# B&R Automation Studio project Get_Weather
Automation Studio 4.2.1.211

## Logical view

### WeaTypes.typ
```iecst
TYPE
	weather_typ : 	STRUCT
		temp : REAL;
		humidity : REAL;
		wind_speed : REAL;
		wind_dir : REAL;
		clouds : REAL;
		isValid : BOOL;
	END_STRUCT;
END_TYPE
```

### WeaVariables.var
```iecst
VAR
	weather : weather_typ;
	response_JSON_valid : BOOL;
	response_JSON : STRING[1000];
END_VAR
```

### Program Logical/GetWeather/doHTTP (IEC)

#### Cyclic.fbd - Cyclic code
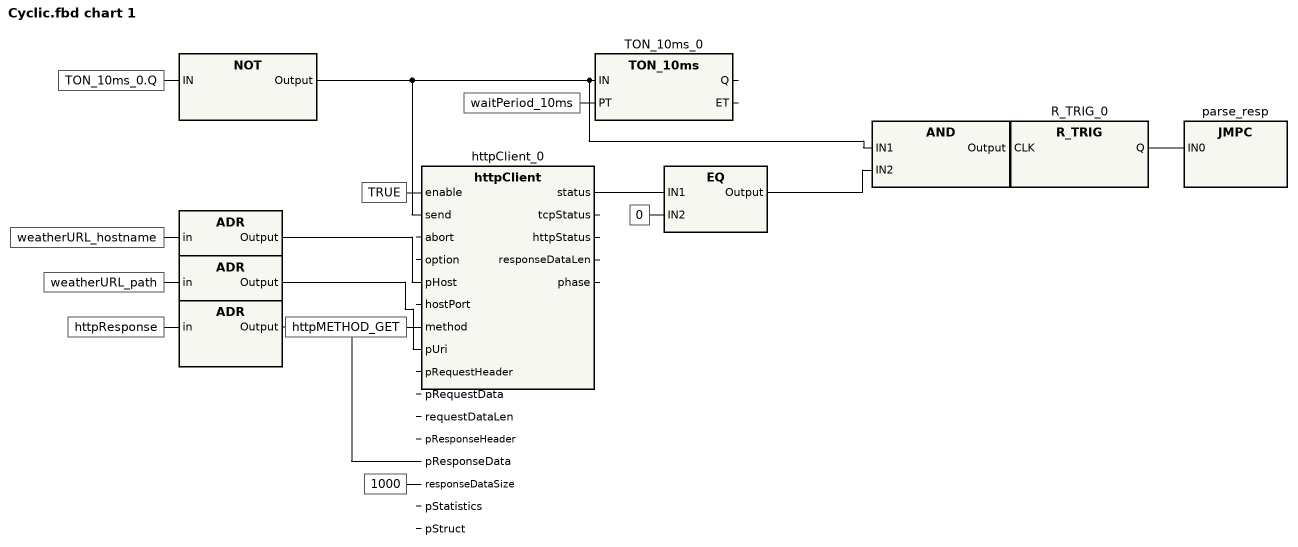
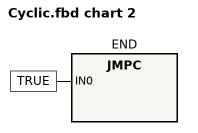
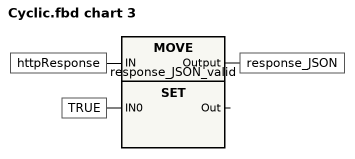
Diagram, in the editor's own instruction-list form stored in the file:
```il
PROGRAM _CYCLIC
VAR
	zz0000FCT_1_1_NOT_Output : ANY;
	zz0000FCT_1_1_ADR_Output : UDINT;
	zz0000FCT_1_2_ADR_Output : UDINT;
	zz0000FCT_1_3_ADR_Output : UDINT;
	zz0000FCT_1_1_EQ_Output : BOOL;
	zz0000FCT_1_1_AND_Output : BOOL;
	zz0000OP_3_1_SET_Out : BOOL;
END_VAR

{NetworkNumber := 1}
LD TON_10ms_0.Q
NOT
ST zz0000FCT_1_1_NOT_Output
LD zz0000FCT_1_1_NOT_Output
ST TON_10ms_0.IN
LD waitPeriod_10ms
ST TON_10ms_0.PT
CAL TON_10ms_0
LD weatherURL_hostname
ADR
ST zz0000FCT_1_1_ADR_Output
LD weatherURL_path
ADR
ST zz0000FCT_1_2_ADR_Output
LD httpResponse
ADR
ST zz0000FCT_1_3_ADR_Output
LD TRUE
ST httpClient_0.enable
LD zz0000FCT_1_1_NOT_Output
ST httpClient_0.send
LD zz0000FCT_1_1_ADR_Output
ST httpClient_0.pHost
LD httpMETHOD_GET
ST httpClient_0.method
LD zz0000FCT_1_2_ADR_Output
ST httpClient_0.pUri
LD zz0000FCT_1_3_ADR_Output
ST httpClient_0.pResponseData
LD 1000
ST httpClient_0.responseDataSize
CAL httpClient_0
LD httpClient_0.status
EQ 0
ST zz0000FCT_1_1_EQ_Output
LD zz0000FCT_1_1_NOT_Output
AND zz0000FCT_1_1_EQ_Output
ST zz0000FCT_1_1_AND_Output
LD zz0000FCT_1_1_AND_Output
ST R_TRIG_0.CLK
CAL R_TRIG_0
LD R_TRIG_0.Q
JMPC parse_resp

{NetworkNumber := 2}
LD TRUE
JMPC END

parse_resp:
{NetworkNumber := 3}
LD httpResponse
MOVE
ST response_JSON
LD TRUE
S response_JSON_valid
LD  response_JSON_valid
ST zz0000OP_3_1_SET_Out

END:
{NetworkNumber := 4}

END_PROGRAM
```

#### Init.fbd - Initialization code
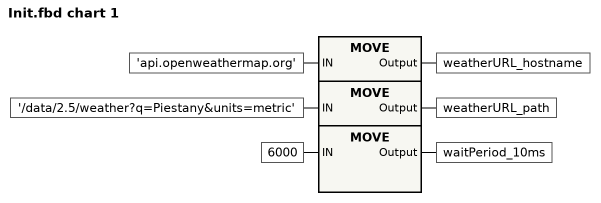
Diagram, in the editor's own instruction-list form stored in the file:
```il
PROGRAM _INIT

{NetworkNumber := 1}
LD 'api.openweathermap.org'
MOVE
ST weatherURL_hostname
LD '/data/2.5/weather?q=Piestany&units=metric'
MOVE
ST weatherURL_path
LD 6000
MOVE
ST waitPeriod_10ms

END_PROGRAM
```

#### Exit.fbd - Exit code
```iecst
PROGRAM _EXIT

(* TODO : Add your code here *)

END_PROGRAM
```

#### GetWheater.var - Local variables
```iecst
VAR
	httpResponse : STRING[1000];
	httpClient_0 : httpClient;
	weatherURL_hostname : STRING[100];
	weatherURL_path : STRING[200];
	TOFF_10ms_0 : TOF_10ms;
	waitPeriod_10ms : UINT;
	R_TRIG_0 : R_TRIG;
	TOF_10ms_0 : TOF_10ms;
	TON_10ms_0 : TON_10ms;
END_VAR
```

### Program Logical/GetWeather/WParser (ANSIC)

#### Cyclic.cpp - Cyclic code
```cpp
#include <bur/plctypes.h>

#ifdef _DEFAULT_INCLUDES
	#include <AsDefault.h>
#endif

#include "jansson.h"

void _CYCLIC ProgramCyclic(void)
{

	if( response_JSON_valid) {
		response_JSON_valid = 0;

		//init structure
		json_t *root;
		json_error_t error;
		root = json_loads(response_JSON, 0, &error);

		if( root) {
			//parse
			/*
			{
			"coord":{"lon":17.75,"lat":48.61},
			"sys":{"message":1.7319,"country":"Slovakia","sunrise":1430623518,"sunset":1430676384},
			"weather":[{"id":500,"main":"Rain","description":"light rain","icon":"10d"}],
			"base":"stations",
			"main":{
			."temp":284.817,
			."temp_min":284.817,
			."temp_max":284.817,
			."pressure":994.66,
			."sea_level":1028.88,
			."grnd_level":994.66,
			."humidity":75},
			"wind":{"speed":3.27,"deg":160.002},
			"clouds":{"all":92},
			"rain":{"3h":0.185},
			"dt":1430646855,
			"id":3056697,
			"name":"Krakovany",
			"cod":200
			}
			*/

			json_t *jmain=json_object_get( root,"main");
			r1=json_unpack(jmain,"{s:F}","temp",&p_temp);
			r2=json_unpack(jmain,"{s:F}","humidity",&p_humidity);

			json_t *jwind=json_object_get( root,"wind");
			r3=json_unpack(jwind,"{s:F}","speed",&p_wind_speed);
			r4=json_unpack(jwind,"{s:F}","deg",&p_wind_deg);

			json_t *jclouds = json_object_get( root,"clouds");
			r5=json_unpack(jclouds,"{s:F}","all",&p_clouds);

			//free
			json_decref(root);

			if( r1+r2+r3+r4+r5 == 0) {
				weather.temp = p_temp;
				weather.clouds = p_clouds;
				weather.wind_dir = p_wind_deg;
				weather.wind_speed = p_wind_speed;
				weather.humidity = p_humidity;
				weather.isValid = 1;
			} else {
				weather.isValid = 0;
			}
		} else { //root not found
			weather.isValid = 0;
		}
	}
}
```

#### Init.cpp - Initialization code
```cpp
#include <bur/plctypes.h>

#ifdef _DEFAULT_INCLUDES
	#include <AsDefault.h>
#endif

void _INIT ProgramInit(void)
{

}
```

#### Exit.cpp - Exit code
```cpp
#include <bur/plctypes.h>

#ifdef _DEFAULT_INCLUDES
	#include <AsDefault.h>
#endif

void _EXIT ProgramExit(void)
{

}
```

#### WParserVar.var - Local variables
```iecst
VAR
	p_humidity : LREAL;
	p_wind_deg : LREAL;
	p_wind_speed : LREAL;
	p_clouds : LREAL;
	r1 : INT;
	r2 : INT;
	r3 : INT;
	r4 : INT;
	r5 : INT;
	p_temp : LREAL;
END_VAR
```

#### hashtable_seed.c
```c
/* Generate sizeof(uint32_t) bytes of as random data as possible to seed
   the hash function.
*/

#ifdef HAVE_CONFIG_H
#include <jansson_private_config.h>
#endif

#include <stdio.h>
#include <time.h>

#ifdef HAVE_STDINT_H
#include <stdint.h>
#endif

#ifdef HAVE_FCNTL_H
#include <fcntl.h>
#endif

#ifdef HAVE_SCHED_H
#include <sched.h>
#endif

#ifdef HAVE_UNISTD_H
#include <unistd.h>
#endif

#ifdef HAVE_SYS_STAT_H
#include <sys/stat.h>
#endif

#ifdef HAVE_SYS_TIME_H
#include <sys/time.h>
#endif

#ifdef HAVE_SYS_TYPES_H
#include <sys/types.h>
#endif

#if defined(_WIN32)
/* For GetModuleHandle(), GetProcAddress() and GetCurrentProcessId() */
#include <windows.h>
#endif

#include "jansson.h"

static uint32_t buf_to_uint32(char *data) {
    size_t i;
    uint32_t result = 0;

    for (i = 0; i < sizeof(uint32_t); i++)
        result = (result << 8) | (unsigned char)data[i];

    return result;
}

/* /dev/urandom */
#if !defined(_WIN32) && defined(USE_URANDOM)
static int seed_from_urandom(uint32_t *seed) {
    /* Use unbuffered I/O if we have open(), close() and read(). Otherwise
       fall back to fopen() */

    char data[sizeof(uint32_t)];
    int ok;

#if defined(HAVE_OPEN) && defined(HAVE_CLOSE) && defined(HAVE_READ)
    int urandom;
    urandom = open("/dev/urandom", O_RDONLY);
    if (urandom == -1)
        return 1;

    ok = read(urandom, data, sizeof(uint32_t)) == sizeof(uint32_t);
    close(urandom);
#else
    FILE *urandom;

    urandom = fopen("/dev/urandom", "rb");
    if (!urandom)
        return 1;

    ok = fread(data, 1, sizeof(uint32_t), urandom) == sizeof(uint32_t);
    fclose(urandom);
#endif

    if (!ok)
        return 1;

    *seed = buf_to_uint32(data);
    return 0;
}
#endif

/* Windows Crypto API */
#if defined(_WIN32) && defined(USE_WINDOWS_CRYPTOAPI)
#include <wincrypt.h>

typedef BOOL (WINAPI *CRYPTACQUIRECONTEXTA)(HCRYPTPROV *phProv, LPCSTR pszContainer, LPCSTR pszProvider, DWORD dwProvType, DWORD dwFlags);
typedef BOOL (WINAPI *CRYPTGENRANDOM)(HCRYPTPROV hProv, DWORD dwLen, BYTE *pbBuffer);
typedef BOOL (WINAPI *CRYPTRELEASECONTEXT)(HCRYPTPROV hProv, DWORD dwFlags);

static int seed_from_windows_cryptoapi(uint32_t *seed)
{
    HINSTANCE hAdvAPI32 = NULL;
    CRYPTACQUIRECONTEXTA pCryptAcquireContext = NULL;
    CRYPTGENRANDOM pCryptGenRandom = NULL;
    CRYPTRELEASECONTEXT pCryptReleaseContext = NULL;
    HCRYPTPROV hCryptProv = 0;
    BYTE data[sizeof(uint32_t)];
    int ok;

    hAdvAPI32 = GetModuleHandle(TEXT("advapi32.dll"));
    if(hAdvAPI32 == NULL)
        return 1;

    pCryptAcquireContext = (CRYPTACQUIRECONTEXTA)GetProcAddress(hAdvAPI32, "CryptAcquireContextA");
    if (!pCryptAcquireContext)
        return 1;

    pCryptGenRandom = (CRYPTGENRANDOM)GetProcAddress(hAdvAPI32, "CryptGenRandom");
    if (!pCryptGenRandom)
        return 1;

    pCryptReleaseContext = (CRYPTRELEASECONTEXT)GetProcAddress(hAdvAPI32, "CryptReleaseContext");
    if (!pCryptReleaseContext)
        return 1;

    if (!pCryptAcquireContext(&hCryptProv, NULL, NULL, PROV_RSA_FULL, CRYPT_VERIFYCONTEXT))
        return 1;

    ok = pCryptGenRandom(hCryptProv, sizeof(uint32_t), data);
    pCryptReleaseContext(hCryptProv, 0);

    if (!ok)
        return 1;

    *seed = buf_to_uint32((char *)data);
    return 0;
}
#endif

/* gettimeofday() and getpid() */
#include "AsTime.h"
static int seed_from_timestamp_and_pid(uint32_t *seed) {
#ifdef HAVE_GETTIMEOFDAY
    /* XOR of seconds and microseconds */
    struct timeval tv;
    gettimeofday(&tv, NULL);
    *seed = (uint32_t)tv.tv_sec ^ (uint32_t)tv.tv_usec;
#else
    /* Seconds only */
	*seed = (uint32_t)clock_ms();
#endif

    /* XOR with PID for more randomness */
#if defined(_WIN32)
    *seed ^= (uint32_t)GetCurrentProcessId();
#elif defined(HAVE_GETPID)
    *seed ^= (uint32_t)getpid();
#endif

    return 0;
}

static uint32_t generate_seed() {
    uint32_t seed;
    int done = 0;

#if !defined(_WIN32) && defined(USE_URANDOM)
    if (!done && seed_from_urandom(&seed) == 0)
        done = 1;
#endif

#if defined(_WIN32) && defined(USE_WINDOWS_CRYPTOAPI)
    if (!done && seed_from_windows_cryptoapi(&seed) == 0)
        done = 1;
#endif

    if (!done) {
        /* Fall back to timestamp and PID if no better randomness is
           available */
        seed_from_timestamp_and_pid(&seed);
    }

    /* Make sure the seed is never zero */
    if (seed == 0)
        seed = 1;

    return seed;
}

volatile uint32_t hashtable_seed = 0;

#if defined(HAVE_ATOMIC_BUILTINS) && (defined(HAVE_SCHED_YIELD) || !defined(_WIN32))
static volatile char seed_initialized = 0;

void json_object_seed(size_t seed) {
    uint32_t new_seed = (uint32_t)seed;

    if (hashtable_seed == 0) {
        if (__atomic_test_and_set(&seed_initialized, __ATOMIC_RELAXED) == 0) {
            /* Do the seeding ourselves */
            if (new_seed == 0)
                new_seed = generate_seed();

            __atomic_store_n(&hashtable_seed, new_seed, __ATOMIC_RELEASE);
        } else {
            /* Wait for another thread to do the seeding */
            do {
#ifdef HAVE_SCHED_YIELD
                sched_yield();
#endif
            } while(__atomic_load_n(&hashtable_seed, __ATOMIC_ACQUIRE) == 0);
        }
    }
}
#elif defined(HAVE_SYNC_BUILTINS) && (defined(HAVE_SCHED_YIELD) || !defined(_WIN32))
void json_object_seed(size_t seed) {
    uint32_t new_seed = (uint32_t)seed;

    if (hashtable_seed == 0) {
        if (new_seed == 0) {
            /* Explicit synchronization fences are not supported by the
               __sync builtins, so every thread getting here has to
               generate the seed value.
            */
            new_seed = generate_seed();
        }

        do {
            if (__sync_bool_compare_and_swap(&hashtable_seed, 0, new_seed)) {
                /* We were the first to seed */
                break;
            } else {
                /* Wait for another thread to do the seeding */
#ifdef HAVE_SCHED_YIELD
                sched_yield();
#endif
            }
        } while(hashtable_seed == 0);
    }
}
#elif defined(_WIN32)
static long seed_initialized = 0;
void json_object_seed(size_t seed) {
    uint32_t new_seed = (uint32_t)seed;

    if (hashtable_seed == 0) {
        if (InterlockedIncrement(&seed_initialized) == 1) {
            /* Do the seeding ourselves */
            if (new_seed == 0)
                new_seed = generate_seed();

            hashtable_seed = new_seed;
        } else {
            /* Wait for another thread to do the seeding */
            do {
                SwitchToThread();
            } while (hashtable_seed == 0);
        }
    }
}
#else
/* Fall back to a thread-unsafe version */
void json_object_seed(size_t seed) {
    uint32_t new_seed = (uint32_t)seed;

    if (hashtable_seed == 0) {
        if (new_seed == 0)
            new_seed = generate_seed();

        hashtable_seed = new_seed;
    }
}
#endif
```

#### memory.c
```c
/*
 * Copyright (c) 2009-2014 Petri Lehtinen <petri@digip.org>
 * Copyright (c) 2011-2012 Basile Starynkevitch <basile@starynkevitch.net>
 *
 * Jansson is free software; you can redistribute it and/or modify it
 * under the terms of the MIT license. See LICENSE for details.
 */

#include <stdlib.h>
#include <string.h>

#include "jansson.h"
#include "jansson_private.h"

unsigned long bur_heap_size = 0x4FFF;

/* C89 allows these to be macros */
#undef malloc
#undef free

/* memory function pointers */
static json_malloc_t do_malloc = malloc;
static json_free_t do_free = free;

void *jsonp_malloc(size_t size)
{
    if(!size)
        return NULL;

    return (*do_malloc)(size);
}

void jsonp_free(void *ptr)
{
    if(!ptr)
        return;

    (*do_free)(ptr);
}

char *jsonp_strdup(const char *str)
{
    return jsonp_strndup(str, strlen(str));
}

char *jsonp_strndup(const char *str, size_t len)
{
    char *new_str;

    new_str = jsonp_malloc(len + 1);
    if(!new_str)
        return NULL;

    memcpy(new_str, str, len);
    new_str[len] = '\0';
    return new_str;
}

void json_set_alloc_funcs(json_malloc_t malloc_fn, json_free_t free_fn)
{
    do_malloc = malloc_fn;
    do_free = free_fn;
}
```

#### value.c
```c
/*
 * Copyright (c) 2009-2014 Petri Lehtinen <petri@digip.org>
 *
 * Jansson is free software; you can redistribute it and/or modify
 * it under the terms of the MIT license. See LICENSE for details.
 */

#ifndef _GNU_SOURCE
#define _GNU_SOURCE
#endif

#ifdef HAVE_CONFIG_H
#include <jansson_private_config.h>
#endif

#include <stddef.h>
#include <stdlib.h>
#include <string.h>
#include <math.h>

#ifdef HAVE_STDINT_H
#include <stdint.h>
#endif

#include "jansson.h"
#include "hashtable.h"
#include "jansson_private.h"
#include "utf.h"

/* Work around nonstandard isnan() and isinf() implementations */
#if 0
#ifndef isnan
#ifndef __sun
static JSON_INLINE int isnan(double x) { return x != x; }
#endif
#endif
#ifndef isinf
static JSON_INLINE int isinf(double x) { return !isnan(x) && isnan(x - x); }
#endif
#endif

static JSON_INLINE void json_init(json_t *json, json_type type)
{
    json->type = type;
    json->refcount = 1;
}

/*** object ***/

extern volatile uint32_t hashtable_seed;

json_t *json_object(void)
{
    json_object_t *object = jsonp_malloc(sizeof(json_object_t));
    if(!object)
        return NULL;

    if (!hashtable_seed) {
        /* Autoseed */
        json_object_seed(0);
    }

    json_init(&object->json, JSON_OBJECT);

    if(hashtable_init(&object->hashtable))
    {
        jsonp_free(object);
        return NULL;
    }

    object->serial = 0;
    object->visited = 0;

    return &object->json;
}

static void json_delete_object(json_object_t *object)
{
    hashtable_close(&object->hashtable);
    jsonp_free(object);
}

size_t json_object_size(const json_t *json)
{
    json_object_t *object;

    if(!json_is_object(json))
        return 0;

    object = json_to_object(json);
    return object->hashtable.size;
}

json_t *json_object_get(const json_t *json, const char *key)
{
    json_object_t *object;

    if(!key || !json_is_object(json))
        return NULL;

    object = json_to_object(json);
    return hashtable_get(&object->hashtable, key);
}

int json_object_set_new_nocheck(json_t *json, const char *key, json_t *value)
{
    json_object_t *object;

    if(!value)
        return -1;

    if(!key || !json_is_object(json) || json == value)
    {
        json_decref(value);
        return -1;
    }
    object = json_to_object(json);

    if(hashtable_set(&object->hashtable, key, object->serial++, value))
    {
        json_decref(value);
        return -1;
    }

    return 0;
}

int json_object_set_new(json_t *json, const char *key, json_t *value)
{
    if(!key || !utf8_check_string(key, strlen(key)))
    {
        json_decref(value);
        return -1;
    }

    return json_object_set_new_nocheck(json, key, value);
}

int json_object_del(json_t *json, const char *key)
{
    json_object_t *object;

    if(!key || !json_is_object(json))
        return -1;

    object = json_to_object(json);
    return hashtable_del(&object->hashtable, key);
}

int json_object_clear(json_t *json)
{
    json_object_t *object;

    if(!json_is_object(json))
        return -1;

    object = json_to_object(json);

    hashtable_clear(&object->hashtable);
    object->serial = 0;

    return 0;
}

int json_object_update(json_t *object, json_t *other)
{
    const char *key;
    json_t *value;

    if(!json_is_object(object) || !json_is_object(other))
        return -1;

    json_object_foreach(other, key, value) {
        if(json_object_set_nocheck(object, key, value))
            return -1;
    }

    return 0;
}

int json_object_update_existing(json_t *object, json_t *other)
{
    const char *key;
    json_t *value;

    if(!json_is_object(object) || !json_is_object(other))
        return -1;

    json_object_foreach(other, key, value) {
        if(json_object_get(object, key))
            json_object_set_nocheck(object, key, value);
    }

    return 0;
}

int json_object_update_missing(json_t *object, json_t *other)
{
    const char *key;
    json_t *value;

    if(!json_is_object(object) || !json_is_object(other))
        return -1;

    json_object_foreach(other, key, value) {
        if(!json_object_get(object, key))
            json_object_set_nocheck(object, key, value);
    }

    return 0;
}

void *json_object_iter(json_t *json)
{
    json_object_t *object;

    if(!json_is_object(json))
        return NULL;

    object = json_to_object(json);
    return hashtable_iter(&object->hashtable);
}

void *json_object_iter_at(json_t *json, const char *key)
{
    json_object_t *object;

    if(!key || !json_is_object(json))
        return NULL;

    object = json_to_object(json);
    return hashtable_iter_at(&object->hashtable, key);
}

void *json_object_iter_next(json_t *json, void *iter)
{
    json_object_t *object;

    if(!json_is_object(json) || iter == NULL)
        return NULL;

    object = json_to_object(json);
    return hashtable_iter_next(&object->hashtable, iter);
}

const char *json_object_iter_key(void *iter)
{
    if(!iter)
        return NULL;

    return hashtable_iter_key(iter);
}

json_t *json_object_iter_value(void *iter)
{
    if(!iter)
        return NULL;

    return (json_t *)hashtable_iter_value(iter);
}

int json_object_iter_set_new(json_t *json, void *iter, json_t *value)
{
    if(!json_is_object(json) || !iter || !value)
        return -1;

    hashtable_iter_set(iter, value);
    return 0;
}

void *json_object_key_to_iter(const char *key)
{
    if(!key)
        return NULL;

    return hashtable_key_to_iter(key);
}

static int json_object_equal(json_t *object1, json_t *object2)
{
    const char *key;
    json_t *value1, *value2;

    if(json_object_size(object1) != json_object_size(object2))
        return 0;

    json_object_foreach(object1, key, value1) {
        value2 = json_object_get(object2, key);

        if(!json_equal(value1, value2))
            return 0;
    }

    return 1;
}

static json_t *json_object_copy(json_t *object)
{
    json_t *result;

    const char *key;
    json_t *value;

    result = json_object();
    if(!result)
        return NULL;

    json_object_foreach(object, key, value)
        json_object_set_nocheck(result, key, value);

    return result;
}

static json_t *json_object_deep_copy(const json_t *object)
{
    json_t *result;
    void *iter;

    result = json_object();
    if(!result)
        return NULL;

    /* Cannot use json_object_foreach because object has to be cast
       non-const */
    iter = json_object_iter((json_t *)object);
    while(iter) {
        const char *key;
        const json_t *value;
        key = json_object_iter_key(iter);
        value = json_object_iter_value(iter);

        json_object_set_new_nocheck(result, key, json_deep_copy(value));
        iter = json_object_iter_next((json_t *)object, iter);
    }

    return result;
}

/*** array ***/

json_t *json_array(void)
{
    json_array_t *array = jsonp_malloc(sizeof(json_array_t));
    if(!array)
        return NULL;
    json_init(&array->json, JSON_ARRAY);

    array->entries = 0;
    array->size = 8;

    array->table = jsonp_malloc(array->size * sizeof(json_t *));
    if(!array->table) {
        jsonp_free(array);
        return NULL;
    }

    array->visited = 0;

    return &array->json;
}

static void json_delete_array(json_array_t *array)
{
    size_t i;

    for(i = 0; i < array->entries; i++)
        json_decref(array->table[i]);

    jsonp_free(array->table);
    jsonp_free(array);
}

size_t json_array_size(const json_t *json)
{
    if(!json_is_array(json))
        return 0;

    return json_to_array(json)->entries;
}

json_t *json_array_get(const json_t *json, size_t index)
{
    json_array_t *array;
    if(!json_is_array(json))
        return NULL;
    array = json_to_array(json);

    if(index >= array->entries)
        return NULL;

    return array->table[index];
}

int json_array_set_new(json_t *json, size_t index, json_t *value)
{
    json_array_t *array;

    if(!value)
        return -1;

    if(!json_is_array(json) || json == value)
    {
        json_decref(value);
        return -1;
    }
    array = json_to_array(json);

    if(index >= array->entries)
    {
        json_decref(value);
        return -1;
    }

    json_decref(array->table[index]);
    array->table[index] = value;

    return 0;
}

static void array_move(json_array_t *array, size_t dest,
                       size_t src, size_t count)
{
    memmove(&array->table[dest], &array->table[src], count * sizeof(json_t *));
}

static void array_copy(json_t **dest, size_t dpos,
                       json_t **src, size_t spos,
                       size_t count)
{
    memcpy(&dest[dpos], &src[spos], count * sizeof(json_t *));
}

static json_t **json_array_grow(json_array_t *array,
                                size_t amount,
                                int copy)
{
    size_t new_size;
    json_t **old_table, **new_table;

    if(array->entries + amount <= array->size)
        return array->table;

    old_table = array->table;

    new_size = max(array->size + amount, array->size * 2);
    new_table = jsonp_malloc(new_size * sizeof(json_t *));
    if(!new_table)
        return NULL;

    array->size = new_size;
    array->table = new_table;

    if(copy) {
        array_copy(array->table, 0, old_table, 0, array->entries);
        jsonp_free(old_table);
        return array->table;
    }

    return old_table;
}

int json_array_append_new(json_t *json, json_t *value)
{
    json_array_t *array;

    if(!value)
        return -1;

    if(!json_is_array(json) || json == value)
    {
        json_decref(value);
        return -1;
    }
    array = json_to_array(json);

    if(!json_array_grow(array, 1, 1)) {
        json_decref(value);
        return -1;
    }

    array->table[array->entries] = value;
    array->entries++;

    return 0;
}

int json_array_insert_new(json_t *json, size_t index, json_t *value)
{
    json_array_t *array;
    json_t **old_table;

    if(!value)
        return -1;

    if(!json_is_array(json) || json == value) {
        json_decref(value);
        return -1;
    }
    array = json_to_array(json);

    if(index > array->entries) {
        json_decref(value);
        return -1;
    }

    old_table = json_array_grow(array, 1, 0);
    if(!old_table) {
        json_decref(value);
        return -1;
    }

    if(old_table != array->table) {
        array_copy(array->table, 0, old_table, 0, index);
        array_copy(array->table, index + 1, old_table, index,
                   array->entries - index);
        jsonp_free(old_table);
    }
    else
        array_move(array, index + 1, index, array->entries - index);

    array->table[index] = value;
    array->entries++;

    return 0;
}

int json_array_remove(json_t *json, size_t index)
{
    json_array_t *array;

    if(!json_is_array(json))
        return -1;
    array = json_to_array(json);

    if(index >= array->entries)
        return -1;

    json_decref(array->table[index]);

    /* If we're removing the last element, nothing has to be moved */
    if(index < array->entries - 1)
        array_move(array, index, index + 1, array->entries - index - 1);

    array->entries--;

    return 0;
}

int json_array_clear(json_t *json)
{
    json_array_t *array;
    size_t i;

    if(!json_is_array(json))
        return -1;
    array = json_to_array(json);

    for(i = 0; i < array->entries; i++)
        json_decref(array->table[i]);

    array->entries = 0;
    return 0;
}

int json_array_extend(json_t *json, json_t *other_json)
{
    json_array_t *array, *other;
    size_t i;

    if(!json_is_array(json) || !json_is_array(other_json))
        return -1;
    array = json_to_array(json);
    other = json_to_array(other_json);

    if(!json_array_grow(array, other->entries, 1))
        return -1;

    for(i = 0; i < other->entries; i++)
        json_incref(other->table[i]);

    array_copy(array->table, array->entries, other->table, 0, other->entries);

    array->entries += other->entries;
    return 0;
}

static int json_array_equal(json_t *array1, json_t *array2)
{
    size_t i, size;

    size = json_array_size(array1);
    if(size != json_array_size(array2))
        return 0;

    for(i = 0; i < size; i++)
    {
        json_t *value1, *value2;

        value1 = json_array_get(array1, i);
        value2 = json_array_get(array2, i);

        if(!json_equal(value1, value2))
            return 0;
    }

    return 1;
}

static json_t *json_array_copy(json_t *array)
{
    json_t *result;
    size_t i;

    result = json_array();
    if(!result)
        return NULL;

    for(i = 0; i < json_array_size(array); i++)
        json_array_append(result, json_array_get(array, i));

    return result;
}

static json_t *json_array_deep_copy(const json_t *array)
{
    json_t *result;
    size_t i;

    result = json_array();
    if(!result)
        return NULL;

    for(i = 0; i < json_array_size(array); i++)
        json_array_append_new(result, json_deep_copy(json_array_get(array, i)));

    return result;
}

/*** string ***/

static json_t *string_create(const char *value, size_t len, int own)
{
    char *v;
    json_string_t *string;

    if(!value)
        return NULL;

    if(own)
        v = (char *)value;
    else {
        v = jsonp_strndup(value, len);
        if(!v)
            return NULL;
    }

    string = jsonp_malloc(sizeof(json_string_t));
    if(!string) {
        if(!own)
            jsonp_free(v);
        return NULL;
    }
    json_init(&string->json, JSON_STRING);
    string->value = v;
    string->length = len;

    return &string->json;
}

json_t *json_string_nocheck(const char *value)
{
    if(!value)
        return NULL;

    return string_create(value, strlen(value), 0);
}

json_t *json_stringn_nocheck(const char *value, size_t len)
{
    return string_create(value, len, 0);
}

/* this is private; "steal" is not a public API concept */
json_t *jsonp_stringn_nocheck_own(const char *value, size_t len)
{
    return string_create(value, len, 1);
}

json_t *json_string(const char *value)
{
    if(!value)
        return NULL;

    return json_stringn(value, strlen(value));
}

json_t *json_stringn(const char *value, size_t len)
{
    if(!value || !utf8_check_string(value, len))
        return NULL;

    return json_stringn_nocheck(value, len);
}

const char *json_string_value(const json_t *json)
{
    if(!json_is_string(json))
        return NULL;

    return json_to_string(json)->value;
}

size_t json_string_length(const json_t *json)
{
    if(!json_is_string(json))
        return 0;

    return json_to_string(json)->length;
}

int json_string_set_nocheck(json_t *json, const char *value)
{
    if(!value)
        return -1;

    return json_string_setn_nocheck(json, value, strlen(value));
}

int json_string_setn_nocheck(json_t *json, const char *value, size_t len)
{
    char *dup;
    json_string_t *string;

    if(!json_is_string(json) || !value)
        return -1;

    dup = jsonp_strndup(value, len);
    if(!dup)
        return -1;

    string = json_to_string(json);
    jsonp_free(string->value);
    string->value = dup;
    string->length = len;

    return 0;
}

int json_string_set(json_t *json, const char *value)
{
    if(!value)
        return -1;

    return json_string_setn(json, value, strlen(value));
}

int json_string_setn(json_t *json, const char *value, size_t len)
{
    if(!value || !utf8_check_string(value, len))
        return -1;

    return json_string_setn_nocheck(json, value, len);
}

static void json_delete_string(json_string_t *string)
{
    jsonp_free(string->value);
    jsonp_free(string);
}

static int json_string_equal(json_t *string1, json_t *string2)
{
    json_string_t *s1, *s2;

    if(!json_is_string(string1) || !json_is_string(string2))
        return 0;

    s1 = json_to_string(string1);
    s2 = json_to_string(string2);
    return s1->length == s2->length && !memcmp(s1->value, s2->value, s1->length);
}

static json_t *json_string_copy(const json_t *string)
{
    json_string_t *s;

    if(!json_is_string(string))
        return NULL;

    s = json_to_string(string);
    return json_stringn_nocheck(s->value, s->length);
}

/*** integer ***/

json_t *json_integer(json_int_t value)
{
    json_integer_t *integer = jsonp_malloc(sizeof(json_integer_t));
    if(!integer)
        return NULL;
    json_init(&integer->json, JSON_INTEGER);

    integer->value = value;
    return &integer->json;
}

json_int_t json_integer_value(const json_t *json)
{
    if(!json_is_integer(json))
        return 0;

    return json_to_integer(json)->value;
}

int json_integer_set(json_t *json, json_int_t value)
{
    if(!json_is_integer(json))
        return -1;

    json_to_integer(json)->value = value;

    return 0;
}

static void json_delete_integer(json_integer_t *integer)
{
    jsonp_free(integer);
}

static int json_integer_equal(json_t *integer1, json_t *integer2)
{
    return json_integer_value(integer1) == json_integer_value(integer2);
}

static json_t *json_integer_copy(const json_t *integer)
{
    return json_integer(json_integer_value(integer));
}

/*** real ***/

json_t *json_real(double value)
{
    json_real_t *real;

    if(isnan(value) || isinf(value))
        return NULL;

    real = jsonp_malloc(sizeof(json_real_t));
    if(!real)
        return NULL;
    json_init(&real->json, JSON_REAL);

    real->value = value;
    return &real->json;
}

double json_real_value(const json_t *json)
{
    if(!json_is_real(json))
        return 0;

    return json_to_real(json)->value;
}

int json_real_set(json_t *json, double value)
{
    if(!json_is_real(json) || isnan(value) || isinf(value))
        return -1;

    json_to_real(json)->value = value;

    return 0;
}

static void json_delete_real(json_real_t *real)
{
    jsonp_free(real);
}

static int json_real_equal(json_t *real1, json_t *real2)
{
    return json_real_value(real1) == json_real_value(real2);
}

static json_t *json_real_copy(const json_t *real)
{
    return json_real(json_real_value(real));
}

/*** number ***/

double json_number_value(const json_t *json)
{
    if(json_is_integer(json))
        return (double)json_integer_value(json);
    else if(json_is_real(json))
        return json_real_value(json);
    else
        return 0.0;
}

/*** simple values ***/

json_t *json_true(void)
{
    static json_t the_true = {JSON_TRUE, (size_t)-1};
    return &the_true;
}

json_t *json_false(void)
{
    static json_t the_false = {JSON_FALSE, (size_t)-1};
    return &the_false;
}

json_t *json_null(void)
{
    static json_t the_null = {JSON_NULL, (size_t)-1};
    return &the_null;
}

/*** deletion ***/

void json_delete(json_t *json)
{
    if(json_is_object(json))
        json_delete_object(json_to_object(json));

    else if(json_is_array(json))
        json_delete_array(json_to_array(json));

    else if(json_is_string(json))
        json_delete_string(json_to_string(json));

    else if(json_is_integer(json))
        json_delete_integer(json_to_integer(json));

    else if(json_is_real(json))
        json_delete_real(json_to_real(json));

    /* json_delete is not called for true, false or null */
}

/*** equality ***/

int json_equal(json_t *json1, json_t *json2)
{
    if(!json1 || !json2)
        return 0;

    if(json_typeof(json1) != json_typeof(json2))
        return 0;

    /* this covers true, false and null as they are singletons */
    if(json1 == json2)
        return 1;

    if(json_is_object(json1))
        return json_object_equal(json1, json2);

    if(json_is_array(json1))
        return json_array_equal(json1, json2);

    if(json_is_string(json1))
        return json_string_equal(json1, json2);

    if(json_is_integer(json1))
        return json_integer_equal(json1, json2);

    if(json_is_real(json1))
        return json_real_equal(json1, json2);

    return 0;
}

/*** copying ***/

json_t *json_copy(json_t *json)
{
    if(!json)
        return NULL;

    if(json_is_object(json))
        return json_object_copy(json);

    if(json_is_array(json))
        return json_array_copy(json);

    if(json_is_string(json))
        return json_string_copy(json);

    if(json_is_integer(json))
        return json_integer_copy(json);

    if(json_is_real(json))
        return json_real_copy(json);

    if(json_is_true(json) || json_is_false(json) || json_is_null(json))
        return json;

    return NULL;
}

json_t *json_deep_copy(const json_t *json)
{
    if(!json)
        return NULL;

    if(json_is_object(json))
        return json_object_deep_copy(json);

    if(json_is_array(json))
        return json_array_deep_copy(json);

    /* for the rest of the types, deep copying doesn't differ from
       shallow copying */

    if(json_is_string(json))
        return json_string_copy(json);

    if(json_is_integer(json))
        return json_integer_copy(json);

    if(json_is_real(json))
        return json_real_copy(json);

    if(json_is_true(json) || json_is_false(json) || json_is_null(json))
        return (json_t *)json;

    return NULL;
}
```

#### jansson.h
```c
/*
 * Copyright (c) 2009-2014 Petri Lehtinen <petri@digip.org>
 *
 * Jansson is free software; you can redistribute it and/or modify
 * it under the terms of the MIT license. See LICENSE for details.
 */

#ifndef JANSSON_H
#define JANSSON_H

#include <stdio.h>
#include <stdlib.h>  /* for size_t */
#include <stdarg.h>

#include "jansson_config.h"

/* Including declarations control unit data types and for B&R ANSI C extensions*/
#include <bur/plctypes.h>

typedef USINT uint8_t;
typedef UINT  uint16_t;
typedef UDINT uint32_t;
typedef SINT int8_t;
typedef INT  int16_t;
typedef DINT int32_t;

#ifdef __cplusplus
extern "C" {
#endif

/* version */

#define JANSSON_MAJOR_VERSION  2
#define JANSSON_MINOR_VERSION  7
#define JANSSON_MICRO_VERSION  0

/* Micro version is omitted if it's 0 */
#define JANSSON_VERSION  "2.7"

/* Version as a 3-byte hex number, e.g. 0x010201 == 1.2.1. Use this
   for numeric comparisons, e.g. #if JANSSON_VERSION_HEX >= ... */
#define JANSSON_VERSION_HEX  ((JANSSON_MAJOR_VERSION << 16) |   \
                              (JANSSON_MINOR_VERSION << 8)  |   \
                              (JANSSON_MICRO_VERSION << 0))

/* types */

typedef enum {
    JSON_OBJECT,
    JSON_ARRAY,
    JSON_STRING,
    JSON_INTEGER,
    JSON_REAL,
    JSON_TRUE,
    JSON_FALSE,
    JSON_NULL
} json_type;

typedef struct json_t {
    json_type type;
    size_t refcount;
} json_t;

#ifndef JANSSON_USING_CMAKE /* disabled if using cmake */
#if JSON_INTEGER_IS_LONG_LONG
#ifdef _WIN32
#define JSON_INTEGER_FORMAT "I64d"
#else
#define JSON_INTEGER_FORMAT "lld"
#endif
typedef long long json_int_t;
#else
#define JSON_INTEGER_FORMAT "ld"
typedef long json_int_t;
#endif /* JSON_INTEGER_IS_LONG_LONG */
#endif

#define json_typeof(json)      ((json)->type)
#define json_is_object(json)   ((json) && json_typeof(json) == JSON_OBJECT)
#define json_is_array(json)    ((json) && json_typeof(json) == JSON_ARRAY)
#define json_is_string(json)   ((json) && json_typeof(json) == JSON_STRING)
#define json_is_integer(json)  ((json) && json_typeof(json) == JSON_INTEGER)
#define json_is_real(json)     ((json) && json_typeof(json) == JSON_REAL)
#define json_is_number(json)   (json_is_integer(json) || json_is_real(json))
#define json_is_true(json)     ((json) && json_typeof(json) == JSON_TRUE)
#define json_is_false(json)    ((json) && json_typeof(json) == JSON_FALSE)
#define json_boolean_value     json_is_true
#define json_is_boolean(json)  (json_is_true(json) || json_is_false(json))
#define json_is_null(json)     ((json) && json_typeof(json) == JSON_NULL)

/* construction, destruction, reference counting */

json_t *json_object(void);
json_t *json_array(void);
json_t *json_string(const char *value);
json_t *json_stringn(const char *value, size_t len);
json_t *json_string_nocheck(const char *value);
json_t *json_stringn_nocheck(const char *value, size_t len);
json_t *json_integer(json_int_t value);
json_t *json_real(double value);
json_t *json_true(void);
json_t *json_false(void);
#define json_boolean(val)      ((val) ? json_true() : json_false())
json_t *json_null(void);

static JSON_INLINE
json_t *json_incref(json_t *json)
{
    if(json && json->refcount != (size_t)-1)
        ++json->refcount;
    return json;
}

/* do not call json_delete directly */
void json_delete(json_t *json);

static JSON_INLINE
void json_decref(json_t *json)
{
    if(json && json->refcount != (size_t)-1 && --json->refcount == 0)
        json_delete(json);
}

/* error reporting */

#define JSON_ERROR_TEXT_LENGTH    160
#define JSON_ERROR_SOURCE_LENGTH   80

typedef struct {
    int line;
    int column;
    int position;
    char source[JSON_ERROR_SOURCE_LENGTH];
    char text[JSON_ERROR_TEXT_LENGTH];
} json_error_t;

/* getters, setters, manipulation */

void json_object_seed(size_t seed);
size_t json_object_size(const json_t *object);
json_t *json_object_get(const json_t *object, const char *key);
int json_object_set_new(json_t *object, const char *key, json_t *value);
int json_object_set_new_nocheck(json_t *object, const char *key, json_t *value);
int json_object_del(json_t *object, const char *key);
int json_object_clear(json_t *object);
int json_object_update(json_t *object, json_t *other);
int json_object_update_existing(json_t *object, json_t *other);
int json_object_update_missing(json_t *object, json_t *other);
void *json_object_iter(json_t *object);
void *json_object_iter_at(json_t *object, const char *key);
void *json_object_key_to_iter(const char *key);
void *json_object_iter_next(json_t *object, void *iter);
const char *json_object_iter_key(void *iter);
json_t *json_object_iter_value(void *iter);
int json_object_iter_set_new(json_t *object, void *iter, json_t *value);

#define json_object_foreach(object, key, value) \
    for(key = json_object_iter_key(json_object_iter(object)); \
        key && (value = json_object_iter_value(json_object_key_to_iter(key))); \
        key = json_object_iter_key(json_object_iter_next(object, json_object_key_to_iter(key))))

#define json_array_foreach(array, index, value) \
	for(index = 0; \
		index < json_array_size(array) && (value = json_array_get(array, index)); \
		index++)

static JSON_INLINE
int json_object_set(json_t *object, const char *key, json_t *value)
{
    return json_object_set_new(object, key, json_incref(value));
}

static JSON_INLINE
int json_object_set_nocheck(json_t *object, const char *key, json_t *value)
{
    return json_object_set_new_nocheck(object, key, json_incref(value));
}

static JSON_INLINE
int json_object_iter_set(json_t *object, void *iter, json_t *value)
{
    return json_object_iter_set_new(object, iter, json_incref(value));
}

size_t json_array_size(const json_t *array);
json_t *json_array_get(const json_t *array, size_t index);
int json_array_set_new(json_t *array, size_t index, json_t *value);
int json_array_append_new(json_t *array, json_t *value);
int json_array_insert_new(json_t *array, size_t index, json_t *value);
int json_array_remove(json_t *array, size_t index);
int json_array_clear(json_t *array);
int json_array_extend(json_t *array, json_t *other);

static JSON_INLINE
int json_array_set(json_t *array, size_t ind, json_t *value)
{
    return json_array_set_new(array, ind, json_incref(value));
}

static JSON_INLINE
int json_array_append(json_t *array, json_t *value)
{
    return json_array_append_new(array, json_incref(value));
}

static JSON_INLINE
int json_array_insert(json_t *array, size_t ind, json_t *value)
{
    return json_array_insert_new(array, ind, json_incref(value));
}

const char *json_string_value(const json_t *string);
size_t json_string_length(const json_t *string);
json_int_t json_integer_value(const json_t *integer);
double json_real_value(const json_t *real);
double json_number_value(const json_t *json);

int json_string_set(json_t *string, const char *value);
int json_string_setn(json_t *string, const char *value, size_t len);
int json_string_set_nocheck(json_t *string, const char *value);
int json_string_setn_nocheck(json_t *string, const char *value, size_t len);
int json_integer_set(json_t *integer, json_int_t value);
int json_real_set(json_t *real, double value);

/* pack, unpack */

json_t *json_pack(const char *fmt, ...);
json_t *json_pack_ex(json_error_t *error, size_t flags, const char *fmt, ...);
json_t *json_vpack_ex(json_error_t *error, size_t flags, const char *fmt, va_list ap);

#define JSON_VALIDATE_ONLY  0x1
#define JSON_STRICT         0x2

int json_unpack(json_t *root, const char *fmt, ...);
int json_unpack_ex(json_t *root, json_error_t *error, size_t flags, const char *fmt, ...);
int json_vunpack_ex(json_t *root, json_error_t *error, size_t flags, const char *fmt, va_list ap);

/* equality */

int json_equal(json_t *value1, json_t *value2);

/* copying */

json_t *json_copy(json_t *value);
json_t *json_deep_copy(const json_t *value);

/* decoding */

#define JSON_REJECT_DUPLICATES  0x1
#define JSON_DISABLE_EOF_CHECK  0x2
#define JSON_DECODE_ANY         0x4
#define JSON_DECODE_INT_AS_REAL 0x8
#define JSON_ALLOW_NUL          0x10

typedef size_t (*json_load_callback_t)(void *buffer, size_t buflen, void *data);

json_t *json_loads(const char *input, size_t flags, json_error_t *error);
json_t *json_loadb(const char *buffer, size_t buflen, size_t flags, json_error_t *error);
json_t *json_loadf(FILE *input, size_t flags, json_error_t *error);
json_t *json_load_file(const char *path, size_t flags, json_error_t *error);
json_t *json_load_callback(json_load_callback_t callback, void *data, size_t flags, json_error_t *error);

/* encoding */

#define JSON_MAX_INDENT         0x1F
#define JSON_INDENT(n)          ((n) & JSON_MAX_INDENT)
#define JSON_COMPACT            0x20
#define JSON_ENSURE_ASCII       0x40
#define JSON_SORT_KEYS          0x80
#define JSON_PRESERVE_ORDER     0x100
#define JSON_ENCODE_ANY         0x200
#define JSON_ESCAPE_SLASH       0x400
#define JSON_REAL_PRECISION(n)  (((n) & 0x1F) << 11)

typedef int (*json_dump_callback_t)(const char *buffer, size_t size, void *data);

char *json_dumps(const json_t *json, size_t flags);
int json_dumpf(const json_t *json, FILE *output, size_t flags);
int json_dump_file(const json_t *json, const char *path, size_t flags);
int json_dump_callback(const json_t *json, json_dump_callback_t callback, void *data, size_t flags);

/* custom memory allocation */

typedef void *(*json_malloc_t)(size_t);
typedef void (*json_free_t)(void *);

void json_set_alloc_funcs(json_malloc_t malloc_fn, json_free_t free_fn);

#ifdef __cplusplus
}
#endif

#endif
```

#### jansson_config.h
```c
/*
 * Copyright (c) 2010-2014 Petri Lehtinen <petri@digip.org>
 *
 * Jansson is free software; you can redistribute it and/or modify
 * it under the terms of the MIT license. See LICENSE for details.
 *
 *
 * This file specifies a part of the site-specific configuration for
 * Jansson, namely those things that affect the public API in
 * jansson.h.
 *
 * The configure script copies this file to jansson_config.h and
 * replaces @var@ substitutions by values that fit your system. If you
 * cannot run the configure script, you can do the value substitution
 * by hand.
 */

#ifndef JANSSON_CONFIG_H
#define JANSSON_CONFIG_H

/* If your compiler supports the inline keyword in C, JSON_INLINE is
   defined to `inline', otherwise empty. In C++, the inline is always
   supported. */
#ifdef __cplusplus
#define JSON_INLINE inline
#else
#define JSON_INLINE
#endif

/* If your compiler supports the `long long` type and the strtoll()
   library function, JSON_INTEGER_IS_LONG_LONG is defined to 1,
   otherwise to 0. */
#define JSON_INTEGER_IS_LONG_LONG 0

/* If locale.h and localeconv() are available, define to 1,
   otherwise to 0. */
#define JSON_HAVE_LOCALECONV 0

#endif
```

#### utf.h
```c
/*
 * Copyright (c) 2009-2014 Petri Lehtinen <petri@digip.org>
 *
 * Jansson is free software; you can redistribute it and/or modify
 * it under the terms of the MIT license. See LICENSE for details.
 */

#ifndef UTF_H
#define UTF_H

#ifdef HAVE_CONFIG_H
#include <jansson_private_config.h>
#endif

#ifdef HAVE_STDINT_H
#include <stdint.h>
#endif

#include "jansson.h"

int utf8_encode(int32_t codepoint, char *buffer, size_t *size);

size_t utf8_check_first(char byte);
size_t utf8_check_full(const char *buffer, size_t size, int32_t *codepoint);
const char *utf8_iterate(const char *buffer, size_t size, int32_t *codepoint);

int utf8_check_string(const char *string, size_t length);

#endif
```

#### README.txt
```
Code is used janson library from https://github.com/akheron/jansson/commits/master
commit: d8753db4ace03e8fa317875ab516f2e6e71375ff

Janson Library licence:
-----------------------
Copyright (c) 2009-2014 Petri Lehtinen <petri@digip.org>

Permission is hereby granted, free of charge, to any person obtaining a copy
of this software and associated documentation files (the "Software"), to deal
in the Software without restriction, including without limitation the rights
to use, copy, modify, merge, publish, distribute, sublicense, and/or sell
copies of the Software, and to permit persons to whom the Software is
furnished to do so, subject to the following conditions:

The above copyright notice and this permission notice shall be included in
all copies or substantial portions of the Software.

THE SOFTWARE IS PROVIDED "AS IS", WITHOUT WARRANTY OF ANY KIND, EXPRESS OR
IMPLIED, INCLUDING BUT NOT LIMITED TO THE WARRANTIES OF MERCHANTABILITY,
FITNESS FOR A PARTICULAR PURPOSE AND NONINFRINGEMENT. IN NO EVENT SHALL THE
AUTHORS OR COPYRIGHT HOLDERS BE LIABLE FOR ANY CLAIM, DAMAGES OR OTHER
LIABILITY, WHETHER IN AN ACTION OF CONTRACT, TORT OR OTHERWISE, ARISING FROM,
OUT OF OR IN CONNECTION WITH THE SOFTWARE OR THE USE OR OTHER DEALINGS IN
THE SOFTWARE.

-----------------------
```

### LICENSE.txt
```
Copyright (c) 2015 Vladimir Pekar <vlapek@vlapek.info>

Permission is hereby granted, free of charge, to any person obtaining a copy
of this software and associated documentation files (the "Software"), to deal
in the Software without restriction, including without limitation the rights
to use, copy, modify, merge, publish, distribute, sublicense, and/or sell
copies of the Software, and to permit persons to whom the Software is
furnished to do so, subject to the following conditions:

The above copyright notice and this permission notice shall be included in
all copies or substantial portions of the Software.

THE SOFTWARE IS PROVIDED "AS IS", WITHOUT WARRANTY OF ANY KIND, EXPRESS OR
IMPLIED, INCLUDING BUT NOT LIMITED TO THE WARRANTIES OF MERCHANTABILITY,
FITNESS FOR A PARTICULAR PURPOSE AND NONINFRINGEMENT. IN NO EVENT SHALL THE
AUTHORS OR COPYRIGHT HOLDERS BE LIABLE FOR ANY CLAIM, DAMAGES OR OTHER
LIABILITY, WHETHER IN AN ACTION OF CONTRACT, TORT OR OTHERWISE, ARISING FROM,
OUT OF OR IN CONNECTION WITH THE SOFTWARE OR THE USE OR OTHER DEALINGS IN
THE SOFTWARE.
```

Listed in the project but not available here: Logical/GetWeather/doHTTP/Types.typ, Logical/GetWeather/WParser/Types.typ, Logical/GetWeather/WParser/dump.c, Logical/GetWeather/WParser/error.c, Logical/GetWeather/WParser/hashtable.c, Logical/GetWeather/WParser/load.c, Logical/GetWeather/WParser/pack_unpack.c, Logical/GetWeather/WParser/strbuffer.c, Logical/GetWeather/WParser/strconv.c, Logical/GetWeather/WParser/utf.c, Logical/GetWeather/WParser/hashtable.h, Logical/GetWeather/WParser/jansson_private.h, Logical/GetWeather/WParser/lookup3.h, Logical/GetWeather/WParser/strbuffer.h
